KUKA KRL program: ho_st631_r3_2.src, ho_st631_r3_2.dat

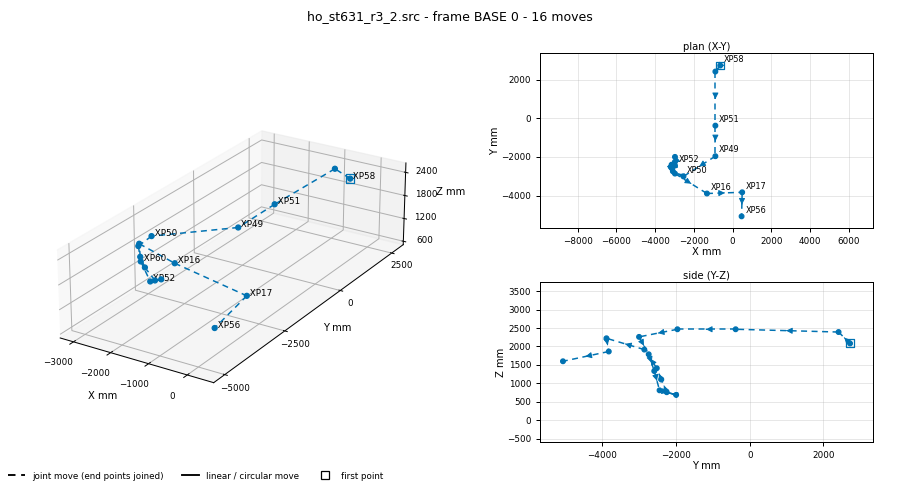
[picture p0: tool path of ho_st631_r3_2.src in frame BASE 0, 16 of 16 moves have a stored position in this frame; points joined in program order, loops and branches not executed]
--- ho_st631_r3_2.src ---
&ACCESS RVO2
&REL 81
&COMMENT Pega lateral ACCELO
&PARAM DISKPATH = KRC:\R1\Program
&PARAM TEMPLATE = C:\KRC\Roboter\Template\vorgabe
&PARAM EDITMASK = *
DEF HO_ST631_R3_2( )
;FOLD INI
  ;FOLD BASISTECH INI
    GLOBAL INTERRUPT DECL 3 WHEN $STOPMESS==TRUE DO IR_STOPM ( )
    INTERRUPT ON 3
    BAS (#INITMOV,0 )
  ;ENDFOLD (BASISTECH INI)
;FOLD GRIPPERTECH INI
USER_GRP(0,DUMMY,DUMMY,GDEFAULT)
;ENDFOLD (GRIPPERTECH INI)
  ;FOLD USER INI
    ;Make your modifications here

  ;ENDFOLD (USER INI)
;ENDFOLD (INI)

; Caracterização dos meios de produção:
; Versão Atual:
; 12/07/2013 12:00 Name: P13.050-R3 CHANGES: Pega Lat. Accelo
; Gripper (F5 6500 0026 579)

chk_w4_wechs_ok ( )       ; CHECK GRIPPER ACCELO

;FOLD PTP P58 CONT Vel=100 % PDAT48 Tool[4]:Gripper Lateral E.Accelo Base[0];%{PE}%R 8.2.20,%MKUKATPBASIS,%CMOVE,%VPTP,%P 1:PTP, 2:P58, 3:C_DIS, 5:100, 7:PDAT48
$BWDSTART=FALSE
PDAT_ACT=PPDAT48
FDAT_ACT=FP58
BAS(#PTP_PARAMS,100)
PTP XP58 C_DIS
;ENDFOLD
;FOLD PTP P48 CONT Vel=100 % PDAT40 Tool[4]:Gripper Lateral E.Accelo Base[0];%{PE}%R 8.2.20,%MKUKATPBASIS,%CMOVE,%VPTP,%P 1:PTP, 2:P48, 3:C_DIS, 5:100, 7:PDAT40
$BWDSTART=FALSE
PDAT_ACT=PPDAT40
FDAT_ACT=FP48
BAS(#PTP_PARAMS,100)
PTP XP48 C_DIS
;ENDFOLD
;FOLD PTP P51 CONT Vel=100 % PDAT43 Tool[4]:Gripper Lateral E.Accelo Base[0];%{PE}%R 8.2.20,%MKUKATPBASIS,%CMOVE,%VPTP,%P 1:PTP, 2:P51, 3:C_DIS, 5:100, 7:PDAT43
$BWDSTART=FALSE
PDAT_ACT=PPDAT43
FDAT_ACT=FP51
BAS(#PTP_PARAMS,100)
PTP XP51 C_DIS
;ENDFOLD
;FOLD PTP P49 Vel=100 % PDAT41 Tool[4]:Gripper Lateral E.Accelo Base[0];%{PE}%R 8.2.20,%MKUKATPBASIS,%CMOVE,%VPTP,%P 1:PTP, 2:P49, 3:, 5:100, 7:PDAT41
$BWDSTART=FALSE
PDAT_ACT=PPDAT41
FDAT_ACT=FP49
BAS(#PTP_PARAMS,100)
PTP XP49
;ENDFOLD

;FOLD OUT 3351 'R3 busca peça Accelo' State=TRUE ;%{PE}%R 8.2.20,%MKUKATPBASIS,%COUT,%VOUTX,%P 2:3351, 3:R3 busca peça Accelo, 5:TRUE, 6:
$OUT[3351]=TRUE
;ENDFOLD
;FOLD WAIT FOR ( IN 3351 'Aguarda Lib. buscar peça Accelo' );%{PE}%R 8.2.20,%MKUKATPBASIS,%CEXT_WAIT_FOR,%VEXT_WAIT_FOR,%P 2:, 4:, 5:$IN, 6:3351, 7:Aguarda Lib. buscar peça Accelo, 9:
WAIT FOR  ( $IN[3351] )
;ENDFOLD
;FOLD OUT 3351 'R3 busca peça Accelo' State=FALSE ;%{PE}%R 8.2.20,%MKUKATPBASIS,%COUT,%VOUTX,%P 2:3351, 3:R3 busca peça Accelo, 5:FALSE, 6:
$OUT[3351]=FALSE
;ENDFOLD

;FOLD PTP P50 CONT Vel=100 % PDAT42 Tool[4]:Gripper Lateral E.Accelo Base[0];%{PE}%R 8.2.20,%MKUKATPBASIS,%CMOVE,%VPTP,%P 1:PTP, 2:P50, 3:C_DIS, 5:100, 7:PDAT42
$BWDSTART=FALSE
PDAT_ACT=PPDAT42
FDAT_ACT=FP50
BAS(#PTP_PARAMS,100)
PTP XP50 C_DIS
;ENDFOLD
;FOLD PTP P61 CONT Vel=100 % PDAT51 Tool[4]:Gripper Lateral E.Accelo Base[0];%{PE}%R 8.2.20,%MKUKATPBASIS,%CMOVE,%VPTP,%P 1:PTP, 2:P61, 3:C_DIS, 5:100, 7:PDAT51
$BWDSTART=FALSE
PDAT_ACT=PPDAT51
FDAT_ACT=FP61
BAS(#PTP_PARAMS,100)
PTP XP61 C_DIS
;ENDFOLD
;FOLD PTP P60 CONT Vel=100 % PDAT50 Tool[4]:Gripper Lateral E.Accelo Base[0];%{PE}%R 8.2.20,%MKUKATPBASIS,%CMOVE,%VPTP,%P 1:PTP, 2:P60, 3:C_DIS, 5:100, 7:PDAT50
$BWDSTART=FALSE
PDAT_ACT=PPDAT50
FDAT_ACT=FP60
BAS(#PTP_PARAMS,100)
PTP XP60 C_DIS
;ENDFOLD
;FOLD PTP P52 CONT Vel=100 % PDAT44 Tool[4]:Gripper Lateral E.Accelo Base[0];%{PE}%R 8.2.20,%MKUKATPBASIS,%CMOVE,%VPTP,%P 1:PTP, 2:P52, 3:C_DIS, 5:100, 7:PDAT44
$BWDSTART=FALSE
PDAT_ACT=PPDAT44
FDAT_ACT=FP52
BAS(#PTP_PARAMS,100)
PTP XP52 C_DIS
;ENDFOLD

;FOLD OUT 3342 'Fora area externa' State=FALSE ;%{PE}%R 8.2.20,%MKUKATPBASIS,%COUT,%VOUTX,%P 2:3342, 3:Fora area externa, 5:FALSE, 6:
$OUT[3342]=FALSE
;ENDFOLD
;FOLD SET Z1 ACCELO State=OPN CONT at START Delay=0 ms;%{PE}%R 8.2.1,%MKUKATPGRP,%CGRP,%VGRP,%P 2:6, 4:1, 5:#YES, 6:GDAT11, 8:0, 10:0
TRIGGER WHEN DISTANCE=0 DELAY=0 DO H50(GRP_APO,6,1,GCONT) PRIO=-1
;ENDFOLD
;FOLD SET Z2 ACCELO State=OPN CONT at START Delay=0 ms;%{PE}%R 8.2.1,%MKUKATPGRP,%CGRP,%VGRP,%P 2:7, 4:1, 5:#YES, 6:GDAT16, 8:0, 10:0
TRIGGER WHEN DISTANCE=0 DELAY=0 DO H50(GRP_APO,7,1,GCONT) PRIO=-1
;ENDFOLD
;FOLD SET Z3 ACCELO State=CONT at START Delay=0 ms;%{PE}%R 8.2.1,%MKUKATPGRP,%CGRP,%VGRP,%P 2:8, 4:1, 5:#YES, 6:GDAT14, 8:0, 10:0
TRIGGER WHEN DISTANCE=0 DELAY=0 DO H50(GRP_APO,8,1,GCONT) PRIO=-1
;ENDFOLD
chk_w4_grp2_opn()
chk_w4_grp1_opn()
chk_w4_grp3_opn()

;FOLD ; POSICAO DE PEGA DA PECA;%{PE}%R 8.2.20,%MKUKATPBASIS,%CCOMMENT,%VNORMAL,%P 2:POSICAO  DE  PEGA  DA  PECA
;ENDFOLD
;FOLD LIN P54 Vel=1 m/s CPDAT31 Tool[4]:Gripper Lateral E.Accelo Base[0];%{PE}%R 8.2.20,%MKUKATPBASIS,%CMOVE,%VLIN,%P 1:LIN, 2:P54, 3:, 5:1, 7:CPDAT31
$BWDSTART=FALSE
LDAT_ACT=LCPDAT31
FDAT_ACT=FP54
BAS(#CP_PARAMS,1)
LIN XP54
;ENDFOLD

IF (NOT(GHOST())) THEN
;FOLD WAIT FOR ( IN 33 'Presença de peça 1 - Accelo' AND IN 34 'Presença de peça 2 - Accelo' );%{PE}%R 8.2.20,%MKUKATPBASIS,%CEXT_WAIT_FOR,%VEXT_WAIT_FOR,%P 2:, 4:, 5:$IN, 6:33, 7:Presença de peça 1 - Accelo, 8:AND, 9:, 10:$IN, 11:34, 12:Presença de peça 2 - Accelo, 14:
WAIT FOR  ( $IN[33] AND $IN[34] )
;ENDFOLD
ENDIF

;FOLD SET Z1 ACCELO State=CLO GDAT7;%{PE}%R 8.2.1,%MKUKATPGRP,%CGRP,%VGRP,%P 2:6, 4:2, 5:#NO, 6:GDAT7, 8:0, 10:0
H50(GRP,6,2,GGDAT7)
;ENDFOLD
chk_w4_grp1_clo()

;FOLD OUT 3350 'R3 solicita liberação p/ sair magazine' State=TRUE ;%{PE}%R 8.2.20,%MKUKATPBASIS,%COUT,%VOUTX,%P 2:3350, 3:R3 solicita liberação p/ sair magazine, 5:TRUE, 6:
$OUT[3350]=TRUE
;ENDFOLD
;FOLD WAIT FOR ( IN 3349 'Aguarda Lib. sair magazine' );%{PE}%R 8.2.20,%MKUKATPBASIS,%CEXT_WAIT_FOR,%VEXT_WAIT_FOR,%P 2:, 4:, 5:$IN, 6:3349, 7:Aguarda Lib. sair magazine, 9:
WAIT FOR  ( $IN[3349] )
;ENDFOLD
;FOLD OUT 3350 'R3 solicita liberação p/ sair magazine' State=FALSE ;%{PE}%R 8.2.20,%MKUKATPBASIS,%COUT,%VOUTX,%P 2:3350, 3:R3 solicita liberação p/ sair magazine, 5:FALSE, 6:
$OUT[3350]=FALSE
;ENDFOLD
;FOLD OUT 3349 'R2 pegou peça' State=FALSE ;%{PE}%R 8.2.20,%MKUKATPBASIS,%COUT,%VOUTX,%P 2:3349, 3:R2 pegou peça, 5:FALSE, 6:
$OUT[3349]=FALSE
;ENDFOLD

;FOLD LIN P55 Vel=1 m/s CPDAT32 Tool[4]:Gripper Lateral E.Accelo Base[0];%{PE}%R 8.2.20,%MKUKATPBASIS,%CMOVE,%VLIN,%P 1:LIN, 2:P55, 3:, 5:1, 7:CPDAT32
$BWDSTART=FALSE
LDAT_ACT=LCPDAT32
FDAT_ACT=FP55
BAS(#CP_PARAMS,1)
LIN XP55
;ENDFOLD

IF (NOT(GHOST())) THEN
;FOLD WAIT FOR ( IN 33 'Presença de peça 1 - Accelo' AND IN 34 'Presença de peça 2 - Accelo' );%{PE}%R 8.2.20,%MKUKATPBASIS,%CEXT_WAIT_FOR,%VEXT_WAIT_FOR,%P 2:, 4:, 5:$IN, 6:33, 7:Presença de peça 1 - Accelo, 8:AND, 9:, 10:$IN, 11:34, 12:Presença de peça 2 - Accelo, 14:
WAIT FOR  ( $IN[33] AND $IN[34] )
;ENDFOLD
ENDIF

;FOLD PTP P62 CONT Vel=100 % PDAT52 Tool[4]:Gripper Lateral E.Accelo Base[0];%{PE}%R 8.2.20,%MKUKATPBASIS,%CMOVE,%VPTP,%P 1:PTP, 2:P62, 3:C_DIS, 5:100, 7:PDAT52
$BWDSTART=FALSE
PDAT_ACT=PPDAT52
FDAT_ACT=FP62
BAS(#PTP_PARAMS,100)
PTP XP62 C_DIS
;ENDFOLD
;FOLD PTP P63 CONT Vel=100 % PDAT53 Tool[4]:Gripper Lateral E.Accelo Base[0];%{PE}%R 8.2.20,%MKUKATPBASIS,%CMOVE,%VPTP,%P 1:PTP, 2:P63, 3:C_DIS, 5:100, 7:PDAT53
$BWDSTART=FALSE
PDAT_ACT=PPDAT53
FDAT_ACT=FP63
BAS(#PTP_PARAMS,100)
PTP XP63 C_DIS
;ENDFOLD
;FOLD PTP P13 CONT Vel=100 % PDAT11 Tool[4]:Gripper Lateral E.Accelo Base[0];%{PE}%R 8.2.20,%MKUKATPBASIS,%CMOVE,%VPTP,%P 1:PTP, 2:P13, 3:C_DIS, 5:100, 7:PDAT11
$BWDSTART=FALSE
PDAT_ACT=PPDAT11
FDAT_ACT=FP13
BAS(#PTP_PARAMS,100)
PTP XP13 C_DIS
;ENDFOLD
;FOLD PTP P16 CONT Vel=100 % PDAT13 Tool[4]:Gripper Lateral E.Accelo Base[0];%{PE}%R 8.2.20,%MKUKATPBASIS,%CMOVE,%VPTP,%P 1:PTP, 2:P16, 3:C_DIS, 5:100, 7:PDAT13
$BWDSTART=FALSE
PDAT_ACT=PPDAT13
FDAT_ACT=FP16
BAS(#PTP_PARAMS,100)
PTP XP16 C_DIS
;ENDFOLD
;FOLD PTP P17 CONT Vel=100 % PDAT14 Tool[4]:Gripper Lateral E.Accelo Base[0];%{PE}%R 8.2.20,%MKUKATPBASIS,%CMOVE,%VPTP,%P 1:PTP, 2:P17, 3:C_DIS, 5:100, 7:PDAT14
$BWDSTART=FALSE
PDAT_ACT=PPDAT14
FDAT_ACT=FP17
BAS(#PTP_PARAMS,100)
PTP XP17 C_DIS
;ENDFOLD
;FOLD PTP P56 CONT Vel=100 % PDAT46 Tool[4]:Gripper Lateral E.Accelo Base[0];%{PE}%R 8.2.20,%MKUKATPBASIS,%CMOVE,%VPTP,%P 1:PTP, 2:P56, 3:C_DIS, 5:100, 7:PDAT46
$BWDSTART=FALSE
PDAT_ACT=PPDAT46
FDAT_ACT=FP56
BAS(#PTP_PARAMS,100)
PTP XP56 C_DIS
;ENDFOLD

;FOLD OUT 3349 'R2 pegou peça' State=TRUE ;%{PE}%R 8.2.20,%MKUKATPBASIS,%COUT,%VOUTX,%P 2:3349, 3:R2 pegou peça, 5:TRUE, 6:
$OUT[3349]=TRUE
;ENDFOLD
;FOLD OUT 3342 'Fora area externa' State=TRUE ;%{PE}%R 8.2.20,%MKUKATPBASIS,%COUT,%VOUTX,%P 2:3342, 3:Fora area externa, 5:TRUE, 6:
$OUT[3342]=TRUE
;ENDFOLD

END

--- ho_st631_r3_2.dat ---
&ACCESS RVO2
&REL 81
&COMMENT Pega lateral ACCELO
&PARAM DISKPATH = KRC:\R1\Program
&PARAM TEMPLATE = C:\KRC\Roboter\Template\vorgabe
&PARAM EDITMASK = *
DEFDAT  ho_st631_r3_2
;FOLD EXTERNAL DECLARATIONS;%{PE}%MKUKATPBASIS,%CEXT,%VCOMMON,%P
;FOLD GRIPPERTECH EXT
EXT  H50 (INT  :IN,INT  :IN,INT  :IN,GRP_TYP  :IN )
;ENDFOLD (GRIPPERTECH EXT)
;FOLD SPOTTECH EXT
EXT  USERSPOT (S_COMMAND  :IN,SPOT_TYPE  :IN )
;ENDFOLD (SPOTTECH EXT)
;FOLD BASISTECH EXT;%{PE}%MKUKATPBASIS,%CEXT,%VEXT,%P
EXT  BAS (BAS_COMMAND  :IN,REAL  :IN )
DECL INT SUCCESS
;ENDFOLD (BASISTECH EXT)
;FOLD USER EXT;%{E}%MKUKATPUSER,%CEXT,%VEXT,%P
;Make your modifications here

;ENDFOLD (USER EXT)
;ENDFOLD (EXTERNAL DECLARATIONS)
DECL BASIS_SUGG_T LAST_BASIS={POINT1[] "P63                     ",POINT2[] "P63                     ",CP_PARAMS[] "CPDAT32                 ",PTP_PARAMS[] "PDAT53                  ",CONT[] "C_DIS                   ",CP_VEL[] "1                       ",PTP_VEL[] "100                     ",SYNC_PARAMS[] "SYNCDAT                 ",SPL_NAME[] "S0                      "}
DECL E6POS XP13={X -2975.51392,Y -2863.0979,Z 1915.146,A -154.053406,B 1.47708201,C 99.7925262,S 2,T 34,E1 3031.13208,E2 0.0,E3 0.0,E4 0.0,E5 0.0,E6 0.0}
DECL FDAT FP13={TOOL_NO 4,BASE_NO 0,IPO_FRAME #BASE,POINT2[] " ",TQ_STATE FALSE}
DECL E6POS XP16={X -1322.46802,Y -3892.06104,Z 2222.17505,A -57.29002,B -4.41215706,C 97.5453491,S 2,T 34,E1 1991.66504,E2 0.0,E3 0.0,E4 0.0,E5 0.0,E6 0.0}
DECL FDAT FP16={TOOL_NO 4,BASE_NO 0,IPO_FRAME #BASE,POINT2[] " ",TQ_STATE FALSE}
DECL E6POS XP17={X 498.76181,Y -3829.20801,Z 1863.36597,A 32.0962181,B -3.45643091,C 110.050598,S 6,T 51,E1 1991.66504,E2 0.0,E3 0.0,E4 0.0,E5 0.0,E6 0.0}
DECL FDAT FP17={TOOL_NO 4,BASE_NO 0,IPO_FRAME #BASE,POINT2[] " ",TQ_STATE FALSE}
DECL PDAT PPDAT11={VEL 100.0,ACC 100.0,APO_DIST 100.0,APO_MODE #CDIS}
DECL PDAT PPDAT13={VEL 100.0,ACC 100.0,APO_DIST 100.0,APO_MODE #CDIS}
DECL PDAT PPDAT14={VEL 100.0,ACC 100.0,APO_DIST 100.0,APO_MODE #CDIS}
DECL GRP_SUGG_T LAST_GRP={NUMBER[] "7                       ",STATE[] "1                       ",PARAMS[] "GDAT15                  "}
DECL GRP_TYP GGDAT1={G_APO #NO,GRP_TIME 0.200000003,CTRL #OFF,DLY 0,DST 1}
DECL GRP_TYP GGDAT2={G_APO #NO,GRP_TIME 0.200000003,CTRL #ON,DLY 0,DST 1}
DECL GRP_TYP GGDAT3={G_APO #NO,GRP_TIME 0.200000003,CTRL #ON,DLY 0,DST 1}
DECL GRP_TYP GGDAT4={G_APO #NO,GRP_TIME 0.200000003,CTRL #ON,DLY 0,DST 1}
DECL GRP_TYP GGDAT5={G_APO #NO,GRP_TIME 0.200000003,CTRL #ON,DLY 0,DST 1}
DECL GRP_TYP GGDAT6={G_APO #NO,GRP_TIME 0.200000003,CTRL #ON,DLY 0,DST 1}
DECL GRP_TYP GGDAT7={G_APO #NO,GRP_TIME 2.0,CTRL #ON,DLY 0,DST 1}
DECL GRP_TYP GGDAT8={G_APO #NO,GRP_TIME 0.200000003,CTRL #OFF,DLY 0,DST 1}
DECL GRP_TYP GGDAT9={G_APO #NO,GRP_TIME 0.200000003,CTRL #OFF,DLY 0,DST 1}
DECL GRP_TYP GGDAT10={G_APO #NO,GRP_TIME 0.200000003,CTRL #OFF,DLY 0,DST 1}
DECL GRP_TYP GGDAT11={G_APO #NO,GRP_TIME 0.200000003,CTRL #ON,DLY 0,DST 1}
DECL GRP_TYP GGDAT12={G_APO #NO,GRP_TIME 0.200000003,CTRL #ON,DLY 0,DST 1}
DECL GRP_TYP GGDAT13={G_APO #NO,GRP_TIME 0.200000003,CTRL #ON,DLY 0,DST 1}
DECL GRP_TYP GGDAT14={G_APO #NO,GRP_TIME 0.200000003,CTRL #OFF,DLY 0,DST 1}
DECL GRP_TYP GGDAT15={G_APO #NO,GRP_TIME 0.200000003,CTRL #OFF,DLY 0,DST 1}
DECL GRP_TYP GGDAT16={G_APO #NO,GRP_TIME 0.200000003,CTRL #OFF,DLY 0,DST 1}
DECL E6POS XP48={X -886.25708,Y 2411.99292,Z 2391.91602,A 148.085205,B -42.3337288,C 116.884804,S 2,T 34,E1 -202.935104,E2 0.0,E3 0.0,E4 0.0,E5 0.0,E6 0.0}
DECL FDAT FP48={TOOL_NO 4,BASE_NO 0,IPO_FRAME #BASE,POINT2[] " ",TQ_STATE FALSE}
DECL PDAT PPDAT40={VEL 100.0,ACC 100.0,APO_DIST 0.0,APO_MODE #CDIS}
DECL E6POS XP49={X -886.254211,Y -1964.64404,Z 2467.13403,A 148.0849,B -42.3345108,C 116.885002,S 2,T 34,E1 4173.70215,E2 0.0,E3 0.0,E4 0.0,E5 0.0,E6 0.0}
DECL FDAT FP49={TOOL_NO 4,BASE_NO 0,IPO_FRAME #BASE,POINT2[] " ",TQ_STATE FALSE}
DECL PDAT PPDAT41={VEL 100.0,ACC 100.0,APO_DIST 100.0,APO_MODE #CDIS}
DECL E6POS XP50={X -2534.21509,Y -3006.302,Z 2260.45288,A -146.7733,B -17.4539509,C 107.014297,S 2,T 34,E1 3825.31592,E2 0.0,E3 0.0,E4 0.0,E5 0.0,E6 0.0}
DECL FDAT FP50={TOOL_NO 4,BASE_NO 0,IPO_FRAME #BASE,POINT2[] " ",TQ_STATE FALSE}
DECL PDAT PPDAT42={VEL 100.0,ACC 100.0,APO_DIST 100.0,APO_MODE #CDIS}
DECL E6POS XP51={X -886.254211,Y -383.418488,Z 2467.13403,A 148.0849,B -42.3345108,C 116.885002,S 2,T 34,E1 2592.47705,E2 0.0,E3 0.0,E4 0.0,E5 0.0,E6 0.0}
DECL FDAT FP51={TOOL_NO 4,BASE_NO 0,IPO_FRAME #BASE,POINT2[] " ",TQ_STATE FALSE}
DECL PDAT PPDAT43={VEL 100.0,ACC 100.0,APO_DIST 100.0,APO_MODE #CDIS}
DECL E6POS XP52={X -2974.50708,Y -2449.79395,Z 808.531616,A -179.3022,B 0.00341867097,C 105.201202,S 2,T 34,E1 3596.70996,E2 0.0,E3 0.0,E4 0.0,E5 0.0,E6 0.0}
DECL FDAT FP52={TOOL_NO 4,BASE_NO 0,IPO_FRAME #BASE,POINT2[] " ",TQ_STATE FALSE}
DECL PDAT PPDAT44={VEL 100.0,ACC 100.0,APO_DIST 100.0,APO_MODE #CDIS}
DECL E6POS XP54={X -2975.125,Y -1999.34204,Z 685.247925,A -179.302307,B 0.00408974197,C 105.202202,S 2,T 34,E1 3596.70898,E2 0.0,E3 0.0,E4 0.0,E5 0.0,E6 0.0}
DECL FDAT FP54={TOOL_NO 4,BASE_NO 0,IPO_FRAME #BASE,POINT2[] " ",TQ_STATE FALSE}
DECL LDAT LCPDAT31={VEL 2.0,ACC 100.0,APO_DIST 100.0,APO_FAC 50.0,AXIS_VEL 100.0,AXIS_ACC 100.0,ORI_TYP #VAR,CIRC_TYP #BASE,JERK_FAC 50.0,GEAR_JERK 50.0,EXAX_IGN 0}
DECL E6POS XP55={X -2975.80396,Y -2254.65405,Z 757.464722,A -179.390305,B 0.0193182994,C 105.641197,S 2,T 34,E1 3596.70801,E2 0.0,E3 0.0,E4 0.0,E5 0.0,E6 0.0}
DECL FDAT FP55={TOOL_NO 4,BASE_NO 0,IPO_FRAME #BASE,POINT2[] " ",TQ_STATE FALSE}
DECL LDAT LCPDAT32={VEL 2.0,ACC 100.0,APO_DIST 100.0,APO_FAC 50.0,AXIS_VEL 100.0,AXIS_ACC 100.0,ORI_TYP #VAR,CIRC_TYP #BASE,JERK_FAC 50.0,GEAR_JERK 50.0,EXAX_IGN 0}
DECL E6POS XP56={X 468.258911,Y -5073.25293,Z 1597.86304,A 30.2174892,B -11.2104301,C 119.264,S 6,T 51,E1 3181.00391,E2 0.0,E3 0.0,E4 0.0,E5 0.0,E6 0.0}
DECL FDAT FP56={TOOL_NO 4,BASE_NO 0,IPO_FRAME #BASE,POINT2[] " ",TQ_STATE FALSE}
DECL PDAT PPDAT46={VEL 100.0,ACC 100.0,APO_DIST 100.0,APO_MODE #CDIS}
DECL GRP_TYP GCONT={G_APO #YES,GRP_TIME 0.0,CTRL #OFF,DLY 0,DST 0}
DECL E6POS XP58={X -634.30011,Y 2723.27808,Z 2082.26001,A 87.8634262,B -48.0646782,C -179.7901,S 2,T 34,E1 -202.940704,E2 0.0,E3 0.0,E4 0.0,E5 0.0,E6 0.0}
DECL FDAT FP58={TOOL_NO 4,BASE_NO 0,IPO_FRAME #BASE,POINT2[] " ",TQ_STATE FALSE}
DECL PDAT PPDAT48={VEL 100.0,ACC 100.0,APO_DIST 100.0,APO_MODE #CDIS}
DECL E6POS XP60={X -3129.60596,Y -2593.95093,Z 1332.92297,A -170.351196,B -13.4717102,C 104.730301,S 2,T 34,E1 3693.94312,E2 0.0,E3 0.0,E4 0.0,E5 0.0,E6 0.0}
DECL FDAT FP60={TOOL_NO 4,BASE_NO 0,IPO_FRAME #BASE,POINT2[] " ",TQ_STATE FALSE}
DECL PDAT PPDAT50={VEL 100.0,ACC 100.0,APO_DIST 100.0,APO_MODE #CDIS}
DECL E6POS XP61={X -3082.78491,Y -2744.97803,Z 1787.49402,A -161.669098,B -14.4397602,C 110.843697,S 2,T 34,E1 3756.86108,E2 0.0,E3 0.0,E4 0.0,E5 0.0,E6 0.0}
DECL FDAT FP61={TOOL_NO 4,BASE_NO 0,IPO_FRAME #BASE,POINT2[] " ",TQ_STATE FALSE}
DECL PDAT PPDAT51={VEL 100.0,ACC 100.0,APO_DIST 100.0,APO_MODE #CDIS}
DECL E6POS XP62={X -3149.73193,Y -2403.01611,Z 1102.45801,A -171.727097,B 0.382275909,C 103.956398,S 2,T 34,E1 3428.66699,E2 0.0,E3 0.0,E4 0.0,E5 0.0,E6 0.0}
DECL FDAT FP62={TOOL_NO 4,BASE_NO 0,IPO_FRAME #BASE,POINT2[] " ",TQ_STATE FALSE}
DECL PDAT PPDAT52={VEL 100.0,ACC 100.0,APO_DIST 100.0,APO_MODE #CDIS}
DECL E6POS XP63={X -3189.18604,Y -2525.24902,Z 1409.17896,A -165.467804,B 0.731544912,C 102.516602,S 2,T 34,E1 3289.59692,E2 0.0,E3 0.0,E4 0.0,E5 0.0,E6 0.0}
DECL FDAT FP63={TOOL_NO 4,BASE_NO 0,IPO_FRAME #BASE,POINT2[] " ",TQ_STATE FALSE}
DECL PDAT PPDAT53={VEL 100.0,ACC 100.0,APO_DIST 100.0,APO_MODE #CDIS}
ENDDAT
